(* IEC 61131-3 sources: CodesysTest/alpha/export/PackML/OMAC/Interfaces/IUnitMode.itf, 3 files *)

(* ---- AllowsEntering.m.st ---- *)
(*#-#-#-#-#-#-#-#-#-#---Declaration---#-#-#-#-#-#-#-#-#-#-#-#-#*)

METHOD AllowsEntering : BOOL
VAR_INPUT
	e: PackMLState;
END_VAR

(* ---- Enter.m.st ---- *)
(*#-#-#-#-#-#-#-#-#-#---Declaration---#-#-#-#-#-#-#-#-#-#-#-#-#*)

METHOD Enter : BOOL
VAR_INPUT
	e: PackMLState;
END_VAR

(* ---- NextState.m.st ---- *)
(*#-#-#-#-#-#-#-#-#-#---Declaration---#-#-#-#-#-#-#-#-#-#-#-#-#*)

METHOD NextState : PackMLState
VAR_INPUT
	e: PackMLState;
END_VAR
